KUKA KRL data list: wkz5_off_1_2.dat

&ACCESS RVP
&REL 4
&COMMENT Pega GRIPPER STB Geobox
&PARAM DISKPATH = KRC:\R1\Program
DEFDAT wkz5_off_1_2
;FOLD EXTERNAL DECLARATIONS;FOLD EXTERNAL DECLARATIONS;%{PE}%MKUKATPBASIS,%CEXT,%VCOMMON,%P
;FOLD GRIPPERTECH EXT
EXT  H50 (INT  :IN,INT  :IN,INT  :IN,GRP_TYP  :IN )
;ENDFOLD (GRIPPERTECH EXT)
;FOLD SPOTTECH EXT

;FOLD BASISTECH EXT;%{PE}%MKUKATPBASIS,%CEXT,%VEXT,%P
EXT  BAS (BAS_COMMAND  :IN,REAL  :IN )
DECL INT SUCCESS
;ENDFOLD (BASISTECH EXT)
;FOLD USER EXT;%{E}%MKUKATPUSER,%CEXT,%VEXT,%P
;Make your modifications here

;ENDFOLD (USER EXT)
;ENDFOLD (EXTERNAL DECLARATIONS)
;# ============ START PATH : bh_p13050r1_ltc_02 =============
DECL BASIS_SUGG_T LAST_BASIS={POINT1[] "P0                      ",POINT2[] "P0                      ",CP_PARAMS[] "CPDAT0                  ",PTP_PARAMS[] "PDAT0                   ",CONT[] "                        ",CP_VEL[] "2.0                     ",PTP_VEL[] "100                     ",SYNC_PARAMS[] "SYNCDAT                 ",SPL_NAME[] "S0                      "}
DECL PDAT PPDAT16={VEL 100.0,ACC 100.0,APO_DIST 100.0,APO_MODE #CDIS}
DECL E6POS XP22={X -2533.1311,Y -5807.38184,Z 2345.9541,A -28.7595501,B -75.2944031,C 88.6572113,S 6,T 18,E1 -5664.646,E2 0.0,E3 0.0,E4 0.0,E5 0.0,E6 0.0}
DECL FDAT FP22={TOOL_NO 8,BASE_NO 0,IPO_FRAME #BASE,POINT2[] " ",TQ_STATE FALSE}
DECL LDAT LCPDAT7={VEL 2.0,ACC 100.0,APO_DIST 100.0,APO_FAC 50.0,AXIS_VEL 100.0,AXIS_ACC 100.0,ORI_TYP #VAR,CIRC_TYP #BASE,JERK_FAC 50.0,GEAR_JERK 50.0,EXAX_IGN 0}
DECL E6POS XP24={X -2617.38403,Y -5952.98096,Z 2346.94995,A -28.7601604,B -75.2951279,C 88.6575089,S 6,T 18,E1 -5664.646,E2 0.0,E3 0.0,E4 0.0,E5 0.0,E6 0.0}
DECL FDAT FP24={TOOL_NO 8,BASE_NO 0,IPO_FRAME #BASE,POINT2[] " ",TQ_STATE FALSE}
DECL LDAT LCPDAT8={VEL 2.0,ACC 100.0,APO_DIST 100.0,APO_FAC 50.0,AXIS_VEL 100.0,AXIS_ACC 100.0,ORI_TYP #VAR,CIRC_TYP #BASE,JERK_FAC 50.0,GEAR_JERK 50.0,EXAX_IGN 0}
DECL E6POS XP25={X -2634.83594,Y -5983.13916,Z 2347.15698,A -28.7603893,B -75.2951508,C 88.657692,S 6,T 18,E1 -5664.646,E2 0.0,E3 0.0,E4 0.0,E5 0.0,E6 0.0}
DECL FDAT FP25={TOOL_NO 8,BASE_NO 0,IPO_FRAME #BASE,POINT2[] " ",TQ_STATE FALSE}
DECL E6POS XP33={X 129.839203,Y -4254.354,Z 2361.24805,A 154.253906,B 41.0406189,C -131.178802,S 2,T 2,E1 -2887.98706,E2 0.0,E3 0.0,E4 0.0,E5 0.0,E6 0.0}
DECL FDAT FP33={TOOL_NO 8,BASE_NO 0,IPO_FRAME #BASE,POINT2[] " ",TQ_STATE FALSE}
DECL PDAT PPDAT25={VEL 100.0,ACC 100.0,APO_DIST 100.0,APO_MODE #CDIS}
DECL E6POS XP39={X -1669.30603,Y -5565.84521,Z 2571.81909,A 132.266998,B -47.6072998,C -70.3760529,S 6,T 18,E1 -4615.20508,E2 0.0,E3 0.0,E4 0.0,E5 0.0,E6 0.0}
DECL FDAT FP39={TOOL_NO 8,BASE_NO 0,IPO_FRAME #BASE,POINT2[] " ",TQ_STATE FALSE}
DECL PDAT PPDAT32={VEL 100.0,ACC 100.0,APO_DIST 100.0,APO_MODE #CDIS}
DECL LDAT LCPDAT9={VEL 2.0,ACC 100.0,APO_DIST 100.0,APO_FAC 50.0,AXIS_VEL 100.0,AXIS_ACC 100.0,ORI_TYP #VAR,CIRC_TYP #BASE,JERK_FAC 50.0,GEAR_JERK 50.0,EXAX_IGN 0}
DECL E6POS XP40={X -2241.26294,Y -6412.22412,Z 1916.90698,A -152.805298,B 89.9557495,C -62.57267,S 6,T 18,E1 -5676.68213,E2 0.0,E3 0.0,E4 0.0,E5 0.0,E6 0.0}
DECL FDAT FP40={TOOL_NO 5,BASE_NO 0,IPO_FRAME #BASE,POINT2[] " ",TQ_STATE FALSE}
DECL E6POS XP44={X -2241.20996,Y -5099.71777,Z 1915.82202,A -93.8118362,B 89.694252,C -3.72019196,S 6,T 18,E1 -4388.68408,E2 0.0,E3 0.0,E4 0.0,E5 0.0,E6 0.0}
DECL FDAT FP44={TOOL_NO 5,BASE_NO 0,IPO_FRAME #BASE,POINT2[] " ",TQ_STATE FALSE}
DECL LDAT LCPDAT12={VEL 2.0,ACC 100.0,APO_DIST 100.0,APO_FAC 50.0,AXIS_VEL 100.0,AXIS_ACC 100.0,ORI_TYP #VAR,CIRC_TYP #BASE,JERK_FAC 50.0,GEAR_JERK 50.0,EXAX_IGN 0}
DECL E6POS XP45={X -620.58313,Y -5296.11816,Z 1915.80298,A -91.3383865,B 89.6957397,C -1.23730004,S 6,T 18,E1 -4388.68701,E2 0.0,E3 0.0,E4 0.0,E5 0.0,E6 0.0}
DECL FDAT FP45={TOOL_NO 5,BASE_NO 0,IPO_FRAME #BASE,POINT2[] " ",TQ_STATE FALSE}
DECL LDAT LCPDAT13={VEL 2.0,ACC 100.0,APO_DIST 100.0,APO_FAC 50.0,AXIS_VEL 100.0,AXIS_ACC 100.0,ORI_TYP #VAR,CIRC_TYP #BASE,JERK_FAC 50.0,GEAR_JERK 50.0,EXAX_IGN 0}
DECL E6POS XP46={X -620.457275,Y -5294.53711,Z 1911.42896,A -50.2860909,B 89.816803,C 39.8137894,S 6,T 18,E1 -3723.19995,E2 0.0,E3 0.0,E4 0.0,E5 0.0,E6 0.0}
DECL FDAT FP46={TOOL_NO 5,BASE_NO 0,IPO_FRAME #BASE,POINT2[] " ",TQ_STATE FALSE}
DECL LDAT LCPDAT14={VEL 2.0,ACC 100.0,APO_DIST 100.0,APO_FAC 50.0,AXIS_VEL 100.0,AXIS_ACC 100.0,ORI_TYP #VAR,CIRC_TYP #BASE,JERK_FAC 50.0,GEAR_JERK 50.0,EXAX_IGN 0}
DECL E6POS XP48={X -368.76001,Y -4764.27686,Z 1909.81604,A -35.6250992,B 89.8164597,C 39.8726387,S 6,T 18,E1 -3723.19995,E2 0.0,E3 0.0,E4 0.0,E5 0.0,E6 0.0}
DECL FDAT FP48={TOOL_NO 5,BASE_NO 0,IPO_FRAME #BASE,POINT2[] " ",TQ_STATE FALSE}
DECL LDAT LCPDAT16={VEL 2.0,ACC 100.0,APO_DIST 100.0,APO_FAC 50.0,AXIS_VEL 100.0,AXIS_ACC 100.0,ORI_TYP #VAR,CIRC_TYP #BASE,JERK_FAC 50.0,GEAR_JERK 50.0,EXAX_IGN 0}
DECL E6POS XP49={X -302.494293,Y -4657.30322,Z 1919.69299,A -84.9462585,B 89.3754425,C -19.9960899,S 6,T 18,E1 -3329.56299,E2 0.0,E3 0.0,E4 0.0,E5 0.0,E6 0.0}
DECL FDAT FP49={TOOL_NO 5,BASE_NO 0,IPO_FRAME #BASE,POINT2[] " ",TQ_STATE FALSE}
DECL PDAT PPDAT36={VEL 100.0,ACC 100.0,APO_DIST 100.0,APO_MODE #CDIS}
DECL E6POS XP50={X 120.587196,Y -4459.74219,Z 1897.79504,A -84.5606232,B 89.3761368,C -19.6216393,S 6,T 18,E1 -3098.72412,E2 0.0,E3 0.0,E4 0.0,E5 0.0,E6 0.0}
DECL FDAT FP50={TOOL_NO 5,BASE_NO 0,IPO_FRAME #BASE,POINT2[] " ",TQ_STATE FALSE}
DECL PDAT PPDAT37={VEL 100.0,ACC 100.0,APO_DIST 100.0,APO_MODE #CDIS}
DECL E6POS XP51={X 368.334686,Y -3953.55908,Z 1864.96204,A 147.892899,B 86.6385574,C -159.870193,S 6,T 18,E1 -2423.94897,E2 0.0,E3 0.0,E4 0.0,E5 0.0,E6 0.0}
DECL FDAT FP51={TOOL_NO 5,BASE_NO 0,IPO_FRAME #BASE,POINT2[] " ",TQ_STATE FALSE}
DECL PDAT PPDAT38={VEL 100.0,ACC 100.0,APO_DIST 100.0,APO_MODE #CDIS}
DECL E6POS XP52={X 350.582397,Y -3688.02295,Z 1990.48596,A 156.707199,B 87.605217,C -165.310593,S 6,T 18,E1 -1754.98706,E2 0.0,E3 0.0,E4 0.0,E5 0.0,E6 0.0}
DECL FDAT FP52={TOOL_NO 5,BASE_NO 0,IPO_FRAME #BASE,POINT2[] " ",TQ_STATE FALSE}
DECL PDAT PPDAT39={VEL 100.0,ACC 100.0,APO_DIST 100.0,APO_MODE #CDIS}
DECL E6POS XP67={X 613.165222,Y -2566.59497,Z 2015.06995,A 93.7516708,B 88.0727463,C 105.921204,S 6,T 18,E1 -703.678711,E2 0.0,E3 0.0,E4 0.0,E5 0.0,E6 0.0}
DECL FDAT FP67={TOOL_NO 5,BASE_NO 0,IPO_FRAME #BASE,POINT2[] " ",TQ_STATE FALSE}
DECL PDAT PPDAT54={VEL 100.0,ACC 100.0,APO_DIST 100.0,APO_MODE #CDIS}
DECL E6POS XP68={X 1005.76599,Y -575.013977,Z 3074.59912,A 75.2860489,B -0.499950409,C 92.0437469,S 6,T 50,E1 309.956299,E2 0.0,E3 0.0,E4 0.0,E5 0.0,E6 0.0}
DECL FDAT FP68={TOOL_NO 5,BASE_NO 0,IPO_FRAME #BASE,POINT2[] " ",TQ_STATE FALSE}
DECL PDAT PPDAT55={VEL 100.0,ACC 100.0,APO_DIST 100.0,APO_MODE #CDIS}
DECL E6POS XP69={X 587.102112,Y -1463.36499,Z 2740.43994,A 78.8688583,B 43.7027893,C 93.8178635,S 6,T 18,E1 69.6376724,E2 0.0,E3 0.0,E4 0.0,E5 0.0,E6 0.0}
DECL FDAT FP69={TOOL_NO 5,BASE_NO 0,IPO_FRAME #BASE,POINT2[] " ",TQ_STATE FALSE}
DECL PDAT PPDAT56={VEL 100.0,ACC 100.0,APO_DIST 100.0,APO_MODE #CDIS}
DECL E6POS XP70={X 1140.604,Y -80.7201996,Z 3409.79712,A 67.0254898,B 0.300575703,C 91.1368179,S 6,T 50,E1 358.183594,E2 0.0,E3 0.0,E4 0.0,E5 0.0,E6 0.0}
DECL FDAT FP70={TOOL_NO 5,BASE_NO 0,IPO_FRAME #BASE,POINT2[] " ",TQ_STATE FALSE}
DECL PDAT PPDAT57={VEL 100.0,ACC 100.0,APO_DIST 100.0,APO_MODE #CDIS}
DECL E6POS XP71={X 1208.83606,Y 177.8078,Z 3409.68091,A 79.5957336,B 0.301005006,C 91.1399536,S 6,T 50,E1 358.168915,E2 0.0,E3 0.0,E4 0.0,E5 0.0,E6 0.0}
DECL FDAT FP71={TOOL_NO 5,BASE_NO 0,IPO_FRAME #BASE,POINT2[] " ",TQ_STATE FALSE}
DECL PDAT PPDAT58={VEL 100.0,ACC 100.0,APO_DIST 100.0,APO_MODE #CDIS}
DECL E6POS XP72={X 1287.33997,Y 609.361023,Z 3384.73999,A 81.3659134,B 3.06711411,C 91.2205963,S 6,T 51,E1 358.178009,E2 0.0,E3 0.0,E4 0.0,E5 0.0,E6 0.0}
DECL FDAT FP72={TOOL_NO 5,BASE_NO 0,IPO_FRAME #BASE,POINT2[] " ",TQ_STATE FALSE}
DECL PDAT PPDAT59={VEL 100.0,ACC 100.0,APO_DIST 100.0,APO_MODE #CDIS}
DECL E6POS XP73={X 1332.67102,Y 908.378784,Z 3368.68408,A 81.370079,B 3.06453395,C 91.212677,S 6,T 51,E1 358.176605,E2 0.0,E3 0.0,E4 0.0,E5 0.0,E6 0.0}
DECL FDAT FP73={TOOL_NO 5,BASE_NO 0,IPO_FRAME #BASE,POINT2[] " ",TQ_STATE FALSE}
DECL PDAT PPDAT60={VEL 100.0,ACC 100.0,APO_DIST 100.0,APO_MODE #CDIS}
DECL E6POS XP74={X 1361.85803,Y 1102.63696,Z 3357.96411,A 95.4746017,B 2.67405605,C 91.9352036,S 6,T 51,E1 358.176208,E2 0.0,E3 0.0,E4 0.0,E5 0.0,E6 0.0}
DECL FDAT FP74={TOOL_NO 5,BASE_NO 0,IPO_FRAME #BASE,POINT2[] " ",TQ_STATE FALSE}
DECL PDAT PPDAT61={VEL 100.0,ACC 100.0,APO_DIST 100.0,APO_MODE #CDIS}
DECL E6POS XP75={X 886.331482,Y 1826.62195,Z 3050.0271,A 137.654602,B 37.7747002,C 93.258522,S 6,T 51,E1 358.178009,E2 0.0,E3 0.0,E4 0.0,E5 0.0,E6 0.0}
DECL FDAT FP75={TOOL_NO 5,BASE_NO 0,IPO_FRAME #BASE,POINT2[] " ",TQ_STATE FALSE}
DECL PDAT PPDAT62={VEL 100.0,ACC 100.0,APO_DIST 100.0,APO_MODE #CDIS}
DECL E6POS XP76={X 415.948486,Y 1808.16699,Z 2250.16504,A -110.554604,B 50.4888191,C 177.1772,S 6,T 51,E1 -116.854698,E2 0.0,E3 0.0,E4 0.0,E5 0.0,E6 0.0}
DECL FDAT FP76={TOOL_NO 5,BASE_NO 0,IPO_FRAME #BASE,POINT2[] " ",TQ_STATE FALSE}
DECL PDAT PPDAT63={VEL 100.0,ACC 100.0,APO_DIST 100.0,APO_MODE #CDIS}
DECL E6POS XP88={X 586.916687,Y -1861.28894,Z 2431.81812,A 81.4868927,B 64.344017,C 91.7723236,S 6,T 18,E1 -266.488495,E2 0.0,E3 0.0,E4 0.0,E5 0.0,E6 0.0}
DECL FDAT FP88={TOOL_NO 5,BASE_NO 0,IPO_FRAME #BASE,POINT2[] " ",TQ_STATE FALSE}
DECL PDAT PPDAT71={VEL 100.0,ACC 100.0,APO_DIST 100.0,APO_MODE #CDIS}
DECL E6POS XP98={X 325.359985,Y 1400.07202,Z 2017.724,A -96.5544968,B 74.0398712,C 168.027802,S 6,T 19,E1 -446.242615,E2 0.0,E3 0.0,E4 0.0,E5 0.0,E6 0.0}
DECL FDAT FP98={TOOL_NO 5,BASE_NO 0,IPO_FRAME #BASE,POINT2[] " ",TQ_STATE FALSE}
DECL PDAT PPDAT78={VEL 100.0,ACC 100.0,APO_DIST 100.0,APO_MODE #CDIS}
DECL GRP_SUGG_T LAST_GRP={NUMBER[] "1                       ",STATE[] "1                       ",PARAMS[] "GDAT2                   "}
DECL GRP_TYP GGDAT1={G_APO #NO,GRP_TIME 0.200000003,CTRL #OFF,DLY 0,DST 1}
DECL GRP_TYP GGDAT2={G_APO #NO,GRP_TIME 0.200000003,CTRL #OFF,DLY 0,DST 1}
ENDDAT ;%{PE}%MKUKATPBASIS,%CEXT,%VCOMMON,%P
;FOLD GRIPPERTECH EXT
